// SIMATIC S7-200 project (STEP 7-Micro/WIN), CPU 224XP REL 02.01

SYMBOL_TABLE USUARIO1
up               I0.0     // ascendente
down             I0.1     // descender
reset            I0.2     // reset
bit_cero         Q0.0
bit_uno          Q0.1
bit_dos          Q0.2
bit_tres         Q0.3
bit_cuatro       Q0.4
bit_cinco        Q0.5
bit_seis         Q0.6
END_SYMBOL_TABLE

ORGANIZATION_BLOCK PRINCIPAL:OB1
TITLE=COMENTARIOS DEL PROGRAMA
BEGIN
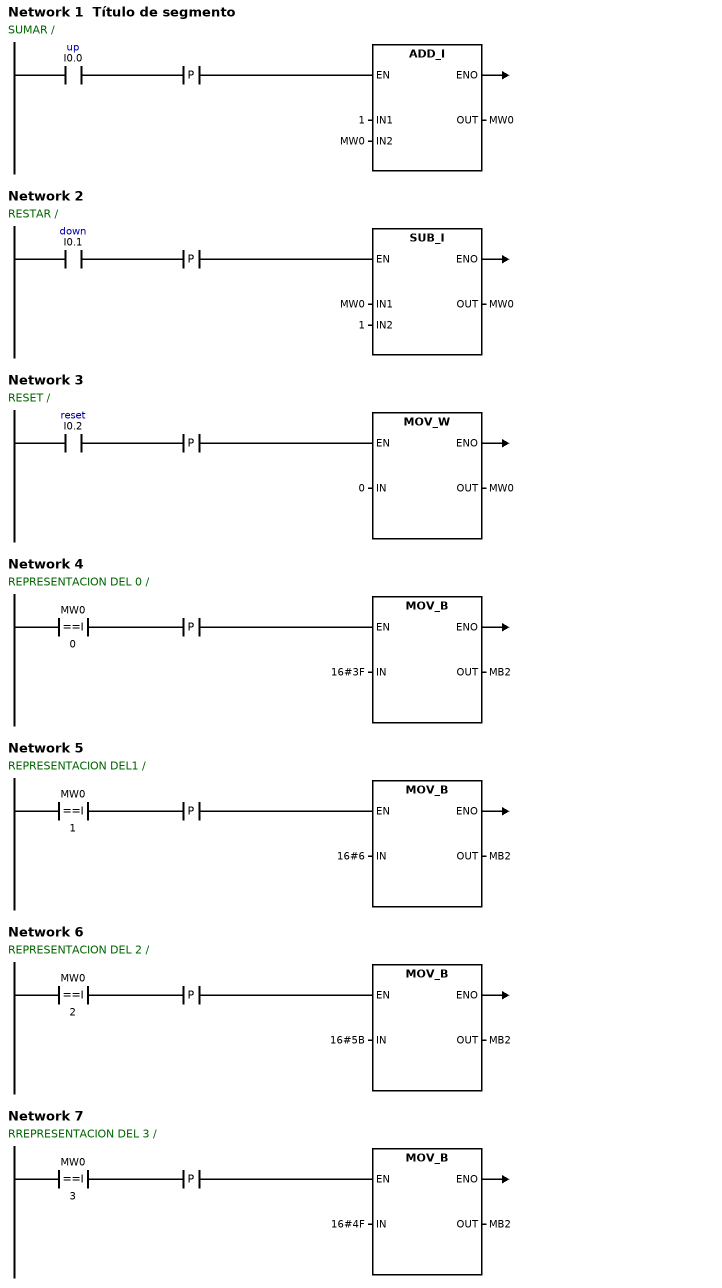
Network 1 // Título de segmento
// SUMAR
// 
LD     up:I0.0
EU
+I     1, MW0
Network 2
// RESTAR
// 
LD     down:I0.1
EU
-I     1, MW0
Network 3
// RESET
// 
LD     reset:I0.2
EU
MOVW   0, MW0
Network 4
// REPRESENTACION DEL 0
// 
// (network saved uncompiled; LAD cells follow)
// row 0: c0 -|==I|- MW0, 0  c1 -|P|-  c2 --  c3 [MOV_B EN:=power@row0, IN:=16#3F, ENO=>power, OUT=>MB2]  c4 ->
// row 1: c3 [box]
Network 5
// REPRESENTACION DEL1
// 
// (network saved uncompiled; LAD cells follow)
// row 0: c0 -|==I|- MW0, 1  c1 -|P|-  c2 --  c3 [MOV_B EN:=power@row0, IN:=16#6, ENO=>power, OUT=>MB2]  c4 ->
// row 1: c3 [box]
Network 6
// REPRESENTACION DEL 2
// 
// (network saved uncompiled; LAD cells follow)
// row 0: c0 -|==I|- MW0, 2  c1 -|P|-  c2 --  c3 [MOV_B EN:=power@row0, IN:=16#5B, ENO=>power, OUT=>MB2]  c4 ->
// row 1: c3 [box]
Network 7
// RREPRESENTACION DEL 3
// 
// (network saved uncompiled; LAD cells follow)
// row 0: c0 -|==I|- MW0, 3  c1 -|P|-  c2 --  c3 [MOV_B EN:=power@row0, IN:=16#4F, ENO=>power, OUT=>MB2]  c4 ->
// row 1: c3 [box]
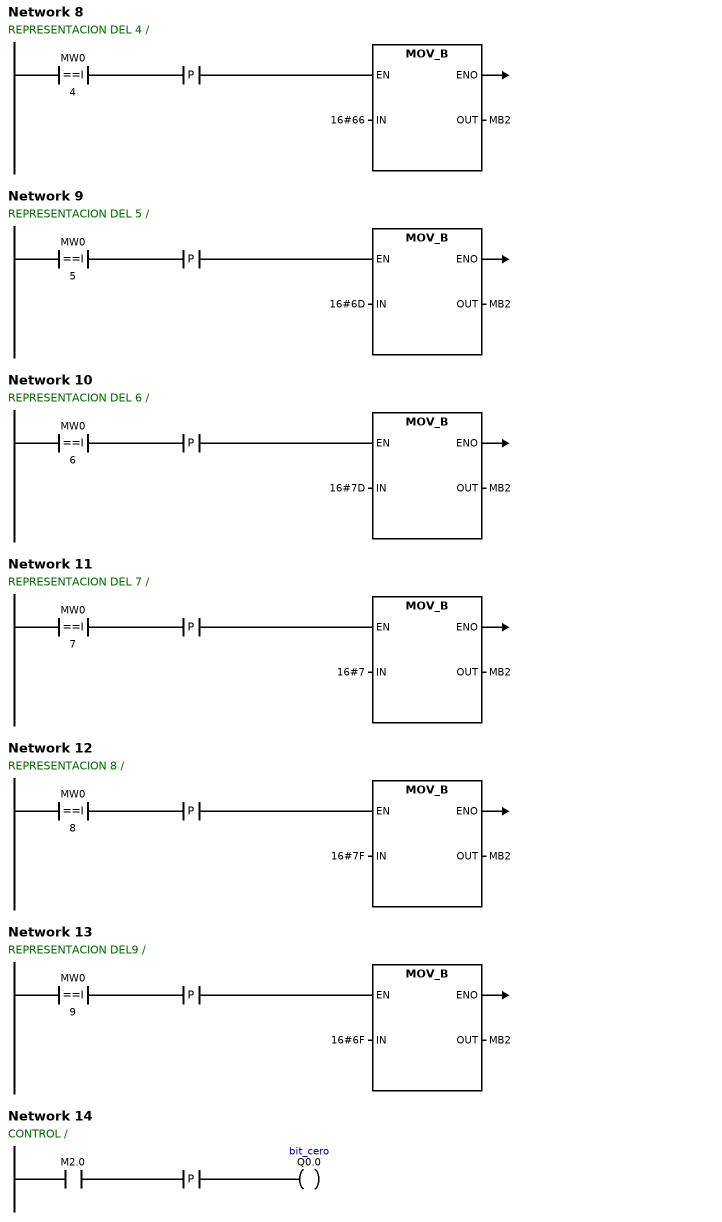
Network 8
// REPRESENTACION DEL 4
// 
// (network saved uncompiled; LAD cells follow)
// row 0: c0 -|==I|- MW0, 4  c1 -|P|-  c2 --  c3 [MOV_B EN:=power@row0, IN:=16#66, ENO=>power, OUT=>MB2]  c4 ->
// row 1: c3 [box]
Network 9
// REPRESENTACION DEL 5
// 
// (network saved uncompiled; LAD cells follow)
// row 0: c0 -|==I|- MW0, 5  c1 -|P|-  c2 --  c3 [MOV_B EN:=power@row0, IN:=16#6D, ENO=>power, OUT=>MB2]  c4 ->
// row 1: c3 [box]
Network 10
// REPRESENTACION DEL 6
// 
// (network saved uncompiled; LAD cells follow)
// row 0: c0 -|==I|- MW0, 6  c1 -|P|-  c2 --  c3 [MOV_B EN:=power@row0, IN:=16#7D, ENO=>power, OUT=>MB2]  c4 ->
// row 1: c3 [box]
Network 11
// REPRESENTACION DEL 7
// 
// (network saved uncompiled; LAD cells follow)
// row 0: c0 -|==I|- MW0, 7  c1 -|P|-  c2 --  c3 [MOV_B EN:=power@row0, IN:=16#7, ENO=>power, OUT=>MB2]  c4 ->
// row 1: c3 [box]
Network 12
// REPRESENTACION 8
// 
// (network saved uncompiled; LAD cells follow)
// row 0: c0 -|==I|- MW0, 8  c1 -|P|-  c2 --  c3 [MOV_B EN:=power@row0, IN:=16#7F, ENO=>power, OUT=>MB2]  c4 ->
// row 1: c3 [box]
Network 13
// REPRESENTACION DEL9
// 
// (network saved uncompiled; LAD cells follow)
// row 0: c0 -|==I|- MW0, 9  c1 -|P|-  c2 --  c3 [MOV_B EN:=power@row0, IN:=16#6F, ENO=>power, OUT=>MB2]  c4 ->
// row 1: c3 [box]
Network 14
// CONTROL
// 
// (network saved uncompiled; LAD cells follow)
// row 0: c0 -| |- M2.0  c1 -|P|-  c2 -( ) bit_cero:Q0.0
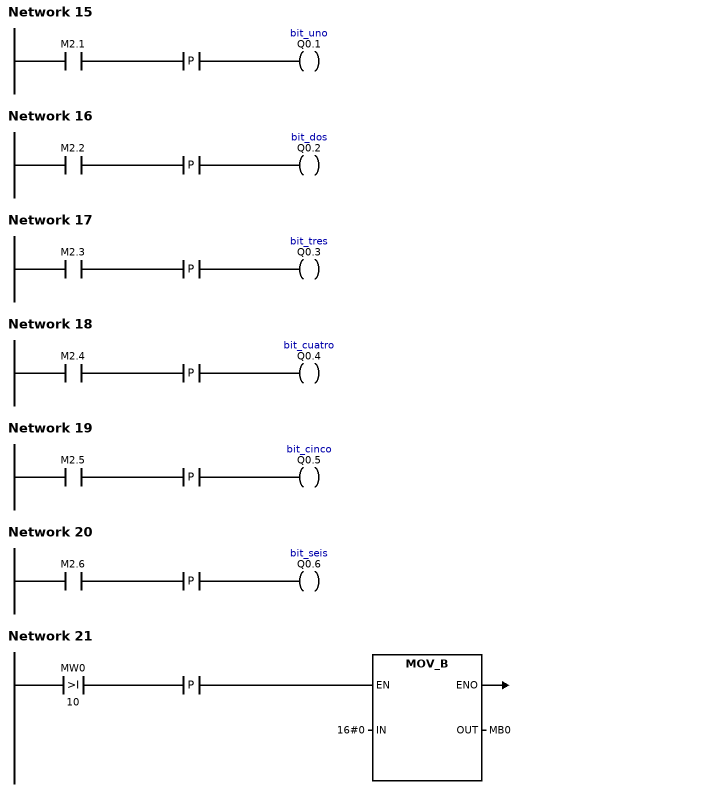
Network 15
// (network saved uncompiled; LAD cells follow)
// row 0: c0 -| |- M2.1  c1 -|P|-  c2 -( ) bit_uno:Q0.1
Network 16
// (network saved uncompiled; LAD cells follow)
// row 0: c0 -| |- M2.2  c1 -|P|-  c2 -( ) bit_dos:Q0.2
Network 17
// (network saved uncompiled; LAD cells follow)
// row 0: c0 -| |- M2.3  c1 -|P|-  c2 -( ) bit_tres:Q0.3
Network 18
// (network saved uncompiled; LAD cells follow)
// row 0: c0 -| |- M2.4  c1 -|P|-  c2 -( ) bit_cuatro:Q0.4
Network 19
// (network saved uncompiled; LAD cells follow)
// row 0: c0 -| |- M2.5  c1 -|P|-  c2 -( ) bit_cinco:Q0.5
Network 20
// (network saved uncompiled; LAD cells follow)
// row 0: c0 -| |- M2.6  c1 -|P|-  c2 -( ) bit_seis:Q0.6
Network 21
LDW>   MW0, 10
EU
MOVB   16#0, MB0
END_ORGANIZATION_BLOCK
